Universal Robots URScript: main.script

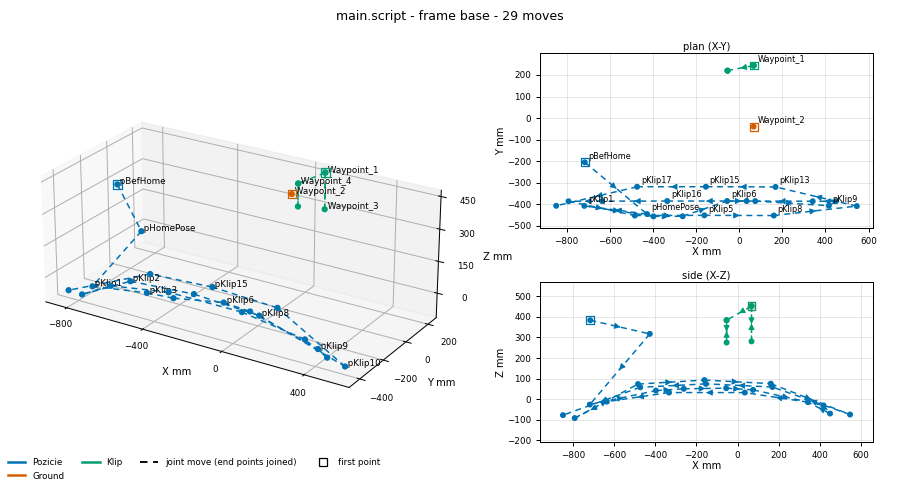
[picture p0: tool path of main.script in frame base, 29 of 29 moves have a stored position in this frame; points joined in program order, loops and branches not executed]
def main():
  set_tcp(p[0.03735271014667435,-0.04548930035733869,0.1890684342738767,0.16978369747036232,0.16108496301516118,1.521587970299213])
  set_payload(0.0, [0.016, 0.0, 0.092])
  step_count_51a1aef3_3718_4bc6_ae28_b8a668176685 = 0.0
  thread Step_Counter_Thread_b15b623d_78f3_454c_ae4b_bda4e6d02093():
    while (True):
      step_count_51a1aef3_3718_4bc6_ae28_b8a668176685 = step_count_51a1aef3_3718_4bc6_ae28_b8a668176685 + 1.0
      sync()
    end
  end
  run Step_Counter_Thread_b15b623d_78f3_454c_ae4b_bda4e6d02093()
  set_tool_voltage(0)
  set_gravity([0.0, 0.0, 9.82])
  set_standard_analog_input_domain(0, 1)
  set_standard_analog_input_domain(1, 1)
  set_tool_analog_input_domain(0, 1)
  set_tool_analog_input_domain(1, 1)
  set_analog_outputdomain(0, 0)
  set_analog_outputdomain(1, 0)
  set_input_actions_to_default()
  set_safety_mode_transition_hardness(1)
  global ipLastPos=p[-0.71904, -0.4068, -0.02549, -2.18405, 2.04498, -0.27993]
  global inPositionNo=1
  def Pozicie():
    $ 10 "Pozicie" "noBreak"
    $ 11 "MoveJ"
    $ 12 "pBefHome" "breakAfter"
    set_tcp(p[0.03735271014667435,-0.04548930035733869,0.1890684342738767,0.16978369747036232,0.16108496301516118,1.521587970299213])
    movej(get_inverse_kin(p[-.715648605996, -.205000950944, .383699304059, -2.203703868463, -.123606847102, 2.189974881807], qnear=[-2.4145699183093186, -1.472981754933496, -2.1753581205950967, -2.660734478627374, -1.0822170416460617, -3.165834013615727]), a=1.3962634015954636, v=1.0471975511965976)
    $ 14 "pHomePose" "breakAfter"
    set_tcp(p[0.03735271014667435,-0.04548930035733869,0.1890684342738767,0.16978369747036232,0.16108496301516118,1.521587970299213])
    movej(get_inverse_kin(p[-.426741112125, -.445008716170, .317531011328, .090042498423, -2.331484726085, 2.036681671981], qnear=[-2.4727817217456227, -1.6048691908465669, -2.008939568196446, -3.1916120688067546, -2.382170263920906, -5.14523703256714]), a=1.3962634015954636, v=1.0471975511965976, r=0.05)
    $ 15 "MoveJ"
    $ 16 "pKlip1" "breakAfter"
    set_tcp(p[0.04,0.02436,0.193,0.1698,0.1611,1.5216])
    movej(get_inverse_kin(p[-.717916350102, -.407007134733, -.025646153500, -2.183732405339, 2.043127291029, -.281934166207], qnear=[-2.4328189531909388, -2.137897316609518, -1.7512834707843226, -0.8102386633502405, -4.675658766423361, -4.019385401402609]), a=3.490658503988659, v=2.0943951023931953)
    $ 17 "pKlip3" "breakAfter"
    set_tcp(p[0.04,0.02436,0.193,0.1698,0.1611,1.5216])
    movej(get_inverse_kin(p[-.397126853785, -.455595776403, .042237014431, -2.246446103699, 2.140231905407, -.081679441001], qnear=[-2.0395086447345134, -1.6564272085772913, -2.3052740732776043, -0.6657837072955672, -4.840316001568938, -3.615596834813251]), a=1.3962634015954636, v=1.0471975511965976)
    $ 18 "pKlip4" "breakAfter"
    set_tcp(p[0.04,0.02436,0.193,0.1698,0.1611,1.5216])
    movej(get_inverse_kin(p[-.261696262434, -.455216130960, .050965765744, -2.246663104422, 2.140151486790, -.081649856141], qnear=[-1.7910898367511194, -1.4943841139422815, -2.437280003224508, -0.728701416646139, -4.856319133435385, -3.365129057561056]), a=1.3962634015954636, v=1.0471975511965976)
    $ 19 "pKlip6" "breakAfter"
    set_tcp(p[0.04,0.02436,0.193,0.1698,0.1611,1.5216])
    movej(get_inverse_kin(p[-.055728808403, -.384407121910, .053915404086, 2.267082870878, -2.158421510344, .001075365499], qnear=[-1.2565210501300257, -1.32275897661318, -2.5424988905536097, -0.8973582426654261, -4.92949098745455, -2.8218005339251917]), a=1.3962634015954636, v=1.0471975511965976)
    $ 20 "pKlip7" "breakAfter"
    set_tcp(p[0.04,0.02436,0.193,0.1698,0.1611,1.5216])
    movej(get_inverse_kin(p[.074794284545, -.384808537956, .045786835457, 2.266807716647, -2.158281213873, .001234201910], qnear=[-0.9635856787310999, -1.3509791533099573, -2.5263879934894007, -0.9454425016986292, -4.9061132113086146, -2.5234525839435022]), a=1.3962634015954636, v=1.0471975511965976)
    $ 21 "pKlip9" "breakAfter"
    set_tcp(p[0.04,0.02436,0.193,0.1698,0.1611,1.5216])
    movej(get_inverse_kin(p[.415981583599, -.406314165961, -.029655193742, 2.048395412832, -1.948348963953, -.407761736493], qnear=[-0.4550259749041956, -1.9097355047809046, -2.060550038014547, -1.3008607069598597, -4.992889467869894, -1.9474733511554163]), a=1.3962634015954636, v=1.0471975511965976)
    $ 23 "pKlip11" "breakAfter"
    set_tcp(p[0.04,0.02436,0.193,0.1698,0.1611,1.5216])
    movej(get_inverse_kin(p[.448509039635, -.385741237724, -.069199723450, -2.176098988853, -2.189923065648, .048969783553], qnear=[-0.3736684958087366, -1.8624690214740198, -2.3984959761248987, -0.31616336504091436, -4.646854702626364, 1.2425787448883057]), a=1.3962634015954636, v=1.0471975511965976)
    $ 24 "pKlip12" "breakAfter"
    set_tcp(p[0.04,0.02436,0.193,0.1698,0.1611,1.5216])
    movej(get_inverse_kin(p[.341020437927, -.385605913533, -.013952595794, -2.152154497266, -2.165384353552, .102578994596], qnear=[-0.44656545320619756, -1.6323545614825647, -2.5015981833087366, -0.4916332403766077, -4.6585344711886805, 1.1688181161880493]), a=1.3962634015954636, v=1.0471975511965976)
    $ 25 "pKlip14" "breakAfter"
    set_tcp(p[0.04,0.02436,0.193,0.1698,0.1611,1.5216])
    movej(get_inverse_kin(p[.034614480199, -.384474368843, .032579285876, -2.188115533390, -2.202644378248, .026097091147], qnear=[-1.0162690321551722, -1.1870186964618128, -2.7012015024768274, -0.7444637457477015, -4.558364335690634, 0.603513240814209]), a=1.3962634015954636, v=1.0471975511965976)
    $ 26 "pKlip16" "breakAfter"
    set_tcp(p[0.04,0.02436,0.193,0.1698,0.1611,1.5216])
    movej(get_inverse_kin(p[-.333422652196, -.384696922539, .032621436167, -2.159257767820, -2.279743429667, -.028168017506], qnear=[-2.048657242451803, -1.5010197798358362, -2.4355302492724817, -0.9018214384662073, -4.53049606481661, -0.4941170851336878]), a=1.3962634015954636, v=1.0471975511965976)
    $ 27 "pKlip18" "breakAfter"
    set_tcp(p[0.04,0.02436,0.193,0.1698,0.1611,1.5216])
    movej(get_inverse_kin(p[-.635306555531, -.385022128679, -.011351189779, 2.089687968229, 2.208175356685, .169234257157], qnear=[-2.4760194460498255, -1.9682586828814905, -1.9280408064471644, -1.1168978849994105, -4.521079126988546, -0.9410370031939905]), a=1.3962634015954636, v=1.0471975511965976)
    $ 28 "pKlip19" "breakAfter"
    set_tcp(p[0.04,0.02436,0.193,0.1698,0.1611,1.5216])
    movej(get_inverse_kin(p[-.791110357619, -.385676933967, -.091336528384, 2.002716311187, 2.116730703607, .340833875748], qnear=[-2.60447866121401, -2.2949731985675257, -1.5290029684649866, -1.3632257620440882, -4.493462983761923, -1.0939739386187952]), a=1.3962634015954636, v=1.0471975511965976)
    $ 29 "MoveJ"
    $ 30 "pKlip2" "breakAfter"
    set_tcp(p[0.03735271014667435,-0.04548930035733869,0.1890684342738767,0.16978369747036232,0.16108496301516118,1.521587970299213])
    movej(get_inverse_kin(p[-.483859358735, -.451883818470, .073893561611, -2.246638894559, 2.140281409628, -.081745850230], qnear=[-2.108490292225973, -1.7756345907794397, -2.0918734709369105, -0.7515171209918421, -4.835193220769064, -3.684976402913229]), a=1.3962634015954636, v=1.0471975511965976)
    $ 31 "pKlip5" "breakAfter"
    set_tcp(p[0.03735271014667435,-0.04548930035733869,0.1890684342738767,0.16978369747036232,0.16108496301516118,1.521587970299213])
    movej(get_inverse_kin(p[-.161364182777, -.450888812909, .093262834498, 2.266833975154, -2.158423850108, .001344525310], qnear=[-1.5223091284381312, -1.444907013569967, -2.3772953192340296, -0.8812463919269007, -4.936122838650839, -3.0939109961139124]), a=1.3962634015954636, v=1.0471975511965976)
    $ 32 "pKlip8" "breakAfter"
    set_tcp(p[0.03735271014667435,-0.04548930035733869,0.1890684342738767,0.16978369747036232,0.16108496301516118,1.521587970299213])
    movej(get_inverse_kin(p[.160789464066, -.451853808286, .075970025419, 2.266603397881, -2.158372721571, .003585999014], qnear=[-0.9005702177630823, -1.479880158101217, -2.352548662816183, -1.0007861296283167, -4.899637166653768, -2.4593947569476526]), a=1.3962634015954636, v=1.0471975511965976)
    $ 33 "pKlip10" "breakAfter"
    set_tcp(p[0.03735271014667435,-0.04548930035733869,0.1890684342738767,0.16978369747036232,0.16108496301516118,1.521587970299213])
    movej(get_inverse_kin(p[.545477499950, -.408071064609, -.073996956338, -.002742154469, -3.132520288529, -.012561900629], qnear=[-0.46371394792665654, -1.931399170552389, -2.2026737372027796, -0.6854804197894495, -4.5262959639178675, -0.42457420030702764]), a=1.3962634015954636, v=1.0471975511965976)
    $ 34 "pKlip13" "breakAfter"
    set_tcp(p[0.03735271014667435,-0.04548930035733869,0.1890684342738767,0.16978369747036232,0.16108496301516118,1.521587970299213])
    movej(get_inverse_kin(p[.168592363322, -.319265413416, .059544992223, -2.188553653104, -2.202614074618, .026892427335], qnear=[-0.5308383146869105, -1.0579512755023401, -2.708611790333883, -0.8023212591754358, -4.613252822552816, 1.0902934074401855]), a=1.3962634015954636, v=1.0471975511965976)
    $ 35 "pKlip15" "breakAfter"
    set_tcp(p[0.03735271014667435,-0.04548930035733869,0.1890684342738767,0.16978369747036232,0.16108496301516118,1.521587970299213])
    movej(get_inverse_kin(p[-.154176956718, -.318207218573, .074987735120, -2.159927318881, -2.279789217327, -.027795055231], qnear=[-1.6401093641864222, -1.024322811757223, -2.645806376134054, -1.0824530760394495, -4.49262518087496, -0.07780105272401983]), a=1.3962634015954636, v=1.0471975511965976)
    $ 36 "pKlip17" "breakAfter"
    set_tcp(p[0.03735271014667435,-0.04548930035733869,0.1890684342738767,0.16978369747036232,0.16108496301516118,1.521587970299213])
    movej(get_inverse_kin(p[-.473001036590, -.318442605685, .058263518914, 2.089628650445, 2.208042346846, .169441286451], qnear=[-2.3946061770068567, -1.63273793855776, -2.2145827452289026, -1.1492322126971644, -4.495126191769735, -0.8608272711383265]), a=1.3962634015954636, v=1.0471975511965976)
    $ 37 "pKlip20" "breakAfter"
    set_tcp(p[0.03735271014667435,-0.04548930035733869,0.1890684342738767,0.16978369747036232,0.16108496301516118,1.521587970299213])
    movej(get_inverse_kin(p[-.848239875745, -.406643074079, -.076967982610, 3.102563228287, .078101539341, .147236896835], qnear=[-2.5431392828570765, -2.240427319203512, -1.6887429396258753, -0.7309921423541468, -4.4598053137408655, 0.6097494959831238]), a=1.3962634015954636, v=1.0471975511965976)
  end
  def Ground():
    $ 38 "Ground" "noBreak"
    $ 39 "Wait: 2.0"
    sleep(2.0)
    $ 40 "MoveJ"
    $ 41 "Waypoint_2" "breakAfter"
    movej(get_inverse_kin(p[.067125472322, -.039538923124, .452728047979, 1.071719089966, 1.761534448119, -1.958523387696], qnear=[1.5507482290267944, -1.1622150580035608, -1.831254784260885, -3.1050623098956507, 1.7321815490722656, -3.8607643286334437]), a=1.3962634015954636, v=1.0471975511965976)
  end
  def Klip():
    $ 42 "Klip" "noBreak"
    $ 43 "MoveJ"
    $ 44 "Waypoint_1" "breakAfter"
    movej(get_inverse_kin(p[.067124251775, .243667209173, .452668543059, 1.071529267825, 1.761357973459, -1.958526259039], qnear=[1.5632219314575195, -1.8334925810443323, -1.212607208882467, -3.0522049109088343, 1.742226243019104, -3.8585458437549036]), a=1.3962634015954636, v=1.0471975511965976)
    $ 45 "MoveJ"
    $ 46 "Waypoint_3" "breakAfter"
    movej(get_inverse_kin(p[.067172056761, .243611856319, .281105485643, 1.071786051218, 1.761605523746, -1.958461394194], qnear=[1.5627070665359497, -1.8820508162127894, -1.5929468313800257, -2.6232274214373987, 1.7419865131378174, -3.859481398259298]), a=1.3962634015954636, v=1.0471975511965976)
    $ 47 "Wait: 1.0"
    sleep(1.0)
    $ 48 "MoveJ"
    $ 49 "Waypoint_1" "breakAfter"
    movej(get_inverse_kin(p[.067124251775, .243667209173, .452668543059, 1.071529267825, 1.761357973459, -1.958526259039], qnear=[1.5632219314575195, -1.8334925810443323, -1.212607208882467, -3.0522049109088343, 1.742226243019104, -3.8585458437549036]), a=1.3962634015954636, v=1.0471975511965976)
    $ 50 "MoveJ"
    $ 51 "Waypoint_4" "breakAfter"
    movej(get_inverse_kin(p[-.053846810550, .219832013324, .383966061240, 1.071526510608, 1.761573970253, -1.958701733627], qnear=[1.8092780113220215, -1.7413232962237757, -1.5024998823748987, -2.8397062460528772, 1.9843173027038574, -3.8100629488574427]), a=1.3962634015954636, v=1.0471975511965976)
    $ 52 "MoveJ"
    $ 53 "Waypoint_5" "breakAfter"
    movej(get_inverse_kin(p[-.053780787706, .219797147073, .275539178358, 1.071641744941, 1.761658226518, -1.958465723906], qnear=[1.8090267181396484, -1.8015311400042933, -1.7142708937274378, -2.567824188862936, 1.9840413331985474, -3.81053072610964]), a=1.3962634015954636, v=1.0471975511965976)
    $ 54 "MoveJ"
    $ 55 "Waypoint_4" "breakAfter"
    movej(get_inverse_kin(p[-.053846810550, .219832013324, .383966061240, 1.071526510608, 1.761573970253, -1.958701733627], qnear=[1.8092780113220215, -1.7413232962237757, -1.5024998823748987, -2.8397062460528772, 1.9843173027038574, -3.8100629488574427]), a=1.3962634015954636, v=1.0471975511965976)
  end
  $ 56 "Thread_1"
  thread Thread_1():
    while (True):
      $ 57 "sync()"
      sync()
      $ 58 "jointPos≔get_actual_joint_positions()"
      global jointPos= get_actual_joint_positions ()
    end
  end
  threadId_Thread_1 = run Thread_1()
  while (True):
    $ 1 "Robot Program"
    $ 2 "pTarget≔p[0,0,0,0,0,0]"
    global pTarget=p[0,0,0,0,0,0]
    $ 3 "nKlipNo≔1"
    global nKlipNo=1
    $ 5 "Script: loop.script"
    def main():
    SetMovementsExtParams()
    while (True):
        global niActionNo = read_input_integer_register(2)
        sync()
    	if (0 == niActionNo):
    		sync()
    	elif (1 == niActionNo):
    		if (read_output_integer_register(2)==255):
                                          Klip()
    	                  end
    	elif (100 == niActionNo):
    		if (read_output_integer_register(2)==255):
    		Ground()
    		end
    	elif (254 == niActionNo):
    		if (read_output_integer_register(2)==255):
    		SetMovementsExtParams ()
    		WriteMovementsExtParams ()
    		end
    	elif (255 == niActionNo):
    		sync()
    	else:
    		popup("nespravne cislo", "Message", False, True, blocking=False)
    		halt
    	end
    	global qActionNumber = niActionNo
    	WriteMovementsExtParams ()
                      sync()
    end
    end
    def SetMovementsExtParams():
        global qActionNumber = read_input_integer_register(2)
        global ActGlobalSpeed=read_input_integer_register(3)
        global ActualToolNmbr=read_input_integer_register(4)
        global ActualWobjNmbr=read_input_integer_register(5)
        global ActualPointNmbr=read_input_integer_register(6)
        global ActUsrSpecSpd1=read_input_float_register(0)
        global ActUsrSpecSpd2=read_input_float_register(1)
        global ActCoordX=read_input_float_register(2)
        global ActCoordY=read_input_float_register(3)
        global ActCoordZ=read_input_float_register(4)
        global ActCoordRx=read_input_float_register(5)
        global ActCoordRy=read_input_float_register(6)
        global ActCoordRz=read_input_float_register(7)
    end
    def WriteMovementsExtParams():
        write_output_integer_register(2, qActionNumber)
        write_output_integer_register(3, ActGlobalSpeed)
        write_output_integer_register(4, ActualToolNmbr)
        write_output_integer_register(5, ActualWobjNmbr)
        write_output_integer_register(6, ActualPointNmbr)
        write_output_float_register(0, ActUsrSpecSpd1)
        write_output_float_register(1, ActUsrSpecSpd2)
        write_output_float_register(2, ActCoordX)
        write_output_float_register(3, ActCoordY)
        write_output_float_register(4, ActCoordZ)
        write_output_float_register(5, ActCoordRx)
        write_output_float_register(6, ActCoordRy)
        write_output_float_register(7, ActCoordRz)
    end
    $ 6 "bTest≔ False "
    global bTest=  False
    $ 9 "main()"
    main()
  end
end
